VAR_GLOBAL CONSTANT
	MAX_OVEN_SEGMENTS 				: UINT := 7;
	MAX_PRINT_HEAD_COUNT			: UINT := 5;
	MAX_PRINT_MODULE_COUNT			: UINT := 2;
END_VAR

(* stored: Version 1.1.0.1, ProductVersion 3.1.0.24
   GVL ItemConst: Id {a686e941-ccd0-44b3-ab18-66c08c56f929} *)
